(* PLC project Senza_nome, Sconosciuto Senza_nome 1 *)
(* stored: creationDateTime 2026-08-24T10:13:13, modificationDateTime 2026-08-24T13:25:29 *)

PROGRAM program0
  VAR
    A1 AT %IX100.0 : BOOL;
    A2 AT %IX100.1 : BOOL;
    Q0 AT %QX100.0 : BOOL;
    A3 AT %IX100.2 : BOOL;
    A4 AT %IX100.3 : BOOL;
    Q1 AT %QX100.1 : BOOL;
    A5 AT %IX100.4 : BOOL;
    A6 AT %IX100.5 : BOOL;
    A7 AT %IX100.6 : BOOL;
    A8 AT %IX100.7 : BOOL;
    Q2 AT %QX100.2 : BOOL;
    A9 AT %IX100.8 : BOOL;
    A10 AT %IX100.9 : BOOL;
    Q3 AT %QX100.3 : BOOL;
    A11 AT %IX100.10 : BOOL;
    A12 AT %IX100.11 : BOOL;
    Q4 AT %QX100.4 : BOOL;
    A13 AT %IX100.12 : BOOL;
    Q5 AT %QX100.5 : BOOL;
  END_VAR

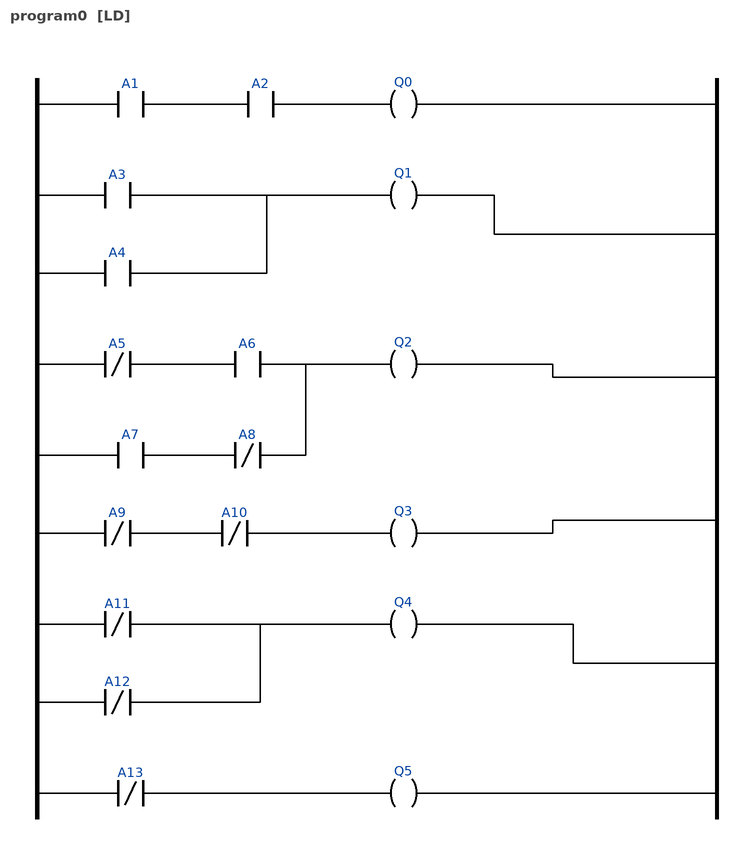
(* LD diagram, written out as Structured Text *)
Q0 := A1 AND A2;
Q1 := A3 OR A4;
Q2 := NOT A5 AND A6 OR A7 AND NOT A8;
Q3 := NOT A9 AND NOT A10;
Q4 := NOT A11 OR NOT A12;
Q5 := NOT A13;
END_PROGRAM

CONFIGURATION Config0
  RESOURCE Res0 ON PLC
    TASK task0(INTERVAL := T#20ms, PRIORITY := 0);
    PROGRAM instance0 WITH task0 : program0;
  END_RESOURCE
END_CONFIGURATION
